TYPE SEND_iCMD_DATA :
STRUCT
	DEVICE_ID       : UDINT;
	FUNCTIONCODE    : UDINT;
	DATA            : LREAL;
	Vel             : LREAL;
END_STRUCT
END_TYPE

(* stored: Version 1.1.0.1, ProductVersion 3.1.4018.5
   DUT SEND_iCMD_DATA: Id {25eeb529-ab31-46d2-888b-815cf06ef658} *)
